TYPE InMotorPDO :
STRUCT
	statusword: UINT;
	fb_position: DINT;
	fb_velocity: DINT;
	fb_op_mode: SINT;
END_STRUCT
END_TYPE

(* stored: Version 1.1.0.1, ProductVersion 3.1.4024.12
   DUT InMotorPDO: Id {fdfff181-66c9-4694-ab18-b085c1bee2d4} *)
